FUNCTION TN_min : real
VAR
	i:DINT;
END_VAR
VAR_IN_OUT
	Inputs: ARRAY[*] OF REAL;
END_VAR

FOR i:=LOWER_BOUND(Inputs,1) TO UPPER_BOUND(Inputs,1) DO
	IF inputs[i] < TN_min THEN
		TN_min:=inputs[i];
	END_IF
END_FOR

END_FUNCTION

(* stored: Version 1.1.0.1, ProductVersion 3.1.4024.6
   POU TN_min: Id {a0d3c5ff-9c13-41b6-ac21-4a99ad469067}, SpecialFunc None *)
